{attribute 'GeneratedUsingTerminal: EL1918-0000-0016'}
{attribute addProperty BoxType "EL1918-0000-0016"}
{attribute addProperty Id "FSLOGIC_InputsFSLOGIC_Inputs_EEE9388E2FSLOGIC_OutputsEMPTY_STRUCTURE0"}
{attribute addProperty CRC "3735766306"}
{attribute addProperty Size "2"}
TYPE Module_2_FSLOGIC_DEAB4522 :
STRUCT
	{attribute addProperty Name "FSLOGIC_Inputs"}
	FSLOGIC_Inputs  : FSLOGIC_Inputs_EEE9388E;
	{attribute addProperty Name "FSLOGIC_Outputs"}
	FSLOGIC_Outputs  : EMPTY_STRUCTURE;
END_STRUCT
END_TYPE

(* stored: Version 1.2.0.0, ProductVersion 3.1.4024.11
   DUT Module_2_FSLOGIC_DEAB4522: Id {2000c49a-69a0-4c90-b1e1-c8c683e7a827} *)
